FUNCTION_BLOCK L0_ReqManager (* Basic Function Block Type *)
  (* Standard: 61499-2 *)
  (* Version 0.0, 2014-09-01, EQUEROL, UJI *)
  (* Version 1.0, 2015-03-03, EQUEROL, UJI *)
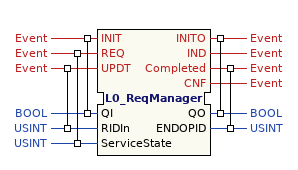
  EVENT_INPUT
    INIT WITH QI; (* Initialization Request *)
    REQ WITH ServiceState; (* Normal Execution Request *)
    UPDT WITH RIDIn; (* Update CNC State *)
  END_EVENT
  EVENT_OUTPUT
    INITO WITH QO; (* Initialization Confirm *)
    IND; (* Service Execution indication *)
    Completed WITH ENDOPID; (* Completed command indication *)
    CNF; (* Execution Confirmation *)
  END_EVENT
  VAR_INPUT
    QI : BOOL; (* Input event qualifier *)
    RIDIn : USINT; (* Execution returned value *)
    ServiceState : USINT; (* Service state *)
  END_VAR
  VAR_OUTPUT
    QO : BOOL; (* Output event qualifier *)
    ENDOPID : USINT; (* Execution returned value *)
  END_VAR
  VAR
    ExecutionRequested : BOOL := FALSE; (* Variable to control if an order was sent *)
  END_VAR
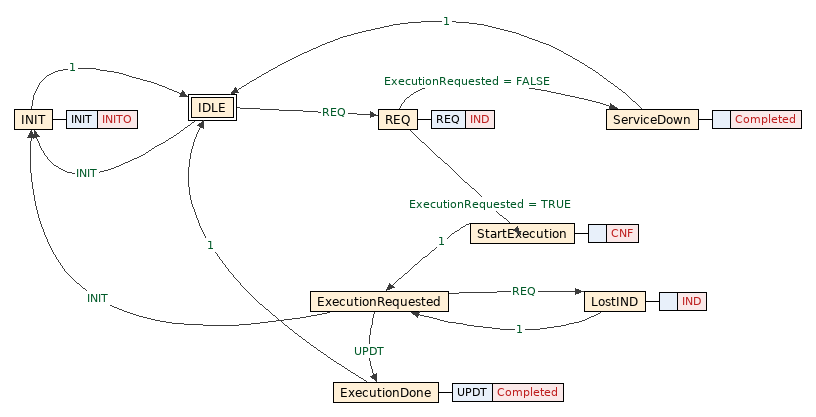
  EC_STATES
    IDLE; (* Initial State *)
    INIT : INIT -> INITO; (* Initialization *)
    REQ : REQ -> IND; (* Normal execution *)
    ExecutionRequested;
    ExecutionDone : UPDT -> Completed;
    ServiceDown : -> Completed;
    StartExecution : -> CNF;
    LostIND : -> IND;
  END_STATES
  EC_TRANSITIONS
    IDLE TO INIT := INIT;
    INIT TO IDLE := 1;
    IDLE TO REQ := REQ;
    ExecutionRequested TO ExecutionDone := UPDT;
    ExecutionDone TO IDLE := 1;
    ExecutionRequested TO INIT := INIT;
    REQ TO ServiceDown := ExecutionRequested = FALSE;
    REQ TO StartExecution := ExecutionRequested = TRUE;
    ServiceDown TO IDLE := 1;
    StartExecution TO ExecutionRequested := 1;
    ExecutionRequested TO LostIND := REQ;
    LostIND TO ExecutionRequested := 1;
  END_TRANSITIONS
  ALGORITHM INIT IN ST: (* Initialization algorithm *)
IF(ExecutionRequested = TRUE) THEN
	ExecutionRequested := FALSE;
	(*TODO: Complete this algorithm to enable service recovery*)
	(*In process action will be lost*)
END_IF;
QO := QI;
  END_ALGORITHM
  ALGORITHM REQ IN ST: (* Normally executed algorithm *)
(*Verify if service is up*)
IF ServiceState =1 THEN
	ExecutionRequested := TRUE;
ELSE
	(*ervice is not up or busy, reject execution request*)
	(*Mark operation as failed but repeatable; TODO: HANDLE the service down case in upper layers*)
	ExecutionRequested := FALSE;
	ENDOPID := 1;
END_IF;
  END_ALGORITHM
  ALGORITHM UPDT IN ST: (* Requested action completed *)
(*TODO: improve error handling, add other states*)
IF RIDIn = 0  THEN
	(*Execution success*)
	ENDOPID := 0;
ELSIF RIDIn= 1 THEN
	(*Execution interrupted*)
	ENDOPID := 1;
ELSE
	(*Execution failed*)
	ENDOPID := 2;
END_IF;
ExecutionRequested := FALSE;
  END_ALGORITHM
END_FUNCTION_BLOCK
